// TIA Portal V20 export
DATA_BLOCK "ControlNodes"   // DB31
AUTHOR : ERsystem_FA2_DH. Kim
// stored: Access Published, MemoryReserve 100, Namespace Unit1
   VAR
      fuses { ExternalWritable := 'False'} : Struct
         motorpower_mcFeedBack : Bool;
         E202CB_motorpower_tripped : Bool;
         E208CB_maincontrol_panelMain_power_tripped : Bool;
         E320CB_E9304PWS_controlpower_SMPS_AC_power_tripped : Bool;
         E326CB_E9404PWS_controlpower_SMPS_AC_power_tripped : Bool;
         E400CB_compensator_X_Axis_power_TR_primarytripped : Bool;
         E410CB_compensator_X_Axis_power_TR_ECONDARYtripped : Bool;
         E500CB_sepa_pnp_X_Axis_powerTr_primary_tripped : Bool;
         E510CB_sepa_pnp_X_Axis_powerTr_ECONDARY_tripped : Bool;
         E720CB_powerMetrt_powerTRIIPED : Bool;
         E726CB_powerMetrt_controlpower_TRIIPED : Bool;
         E3304CB_compensator_X_Axis_power_onTrippred : Bool;
         E3504CB_sepa_pnp1_X_Axis_power_onTrippred : Bool;
         E3604CB_sepa_pnp2_X_Axis_power_onTrippred : Bool;
         E7116CB_procrssor_power_ontrippred : Bool;
         E7156CB_maincontrol_panelHot_power_tripped : Bool;
         E7304CB_panelLed_power_tripped : Bool;
         E8100CB_120VAC_control_powerTr_primary_tripped : Bool;
         E8110CB_120VAC_control_powerTr_secondary_tripped : Bool;
         E8116CB_control_power_ONtripped : Bool;
         E8156CB_maincontrol_panelControl_power_tripped : Bool;
         E9122CB_encoder_terminalUnit_control_power_tripped : Bool;
         E9128CB_servo_control_UNITcontrol_power_tripped : Bool;
         E9204CB_panelFan_power_tripped : Bool;
         E9306CB_controlDc_power_tripped : Bool;
         E9316CB_servo_control_power_tripped : Bool;
         E9406CB_controlDc_power_tripped : Bool;
         E9416CB_junctionBox_class_2SMPS_tripped : Bool;
         E9422CB_EQUIPMENT_LED_power_tripped : Bool;
         E214CB_E6404PWS_controlLER_power_SMPS_AC_power_tripped : Bool;
         E222CB_E6704PWS_controlLER_power_SMPS_AC_power_tripped : Bool;
         E226CB_E6804PWS_safety_power_SMPS_AC_power_tripped : Bool;
         E4120CB_procrssor_power_onTrpped : Bool;
         E4126CB_programing_power_outletTrpped : Bool;
         E4304CB_panelLed_power_tripped : Bool;
         E4420CB_controlLevel_hub_power_tripped : Bool;
         E4426CB_mainHmi_power_tripped : Bool;
         E4432CB_portableHmi_power_TIPPED : Bool;
         E4604CB_panelIrtHub_power_TIPPED : Bool;
         E4608ES_irtHub_fault : Bool;
         E5110CB_120VAC_control_power_TR_secondary_tripped : Bool;
         E5120CB_control_power_onTrippred : Bool;
         E5126CB_visionMonitor1_MCU_power_strip_outlet_power_tripped : Bool;
         E5132CB_visionMonitor2_visionMonitor3_power_strip_outlet_power_tripped : Bool;
         E5156CB_vision_LIGHT_controller_power_strip_outlet_power_tripped : Bool;
         E5222CB_FFU_power1_power_tripped : Bool;
         E6154CB_ET200MP_io_output_power_tripped : Bool;
         E6180CB_junctionBox_control_power_tripped : Bool;
         E6204CB_class2_SMPS_power_tripped : Bool;
         E6220CB_ET200ECO_PN1_power_tripped : Bool;
         E6224CB_ET200ECO_PN2_power_tripped : Bool;
         E6228CB_ET200ECO_PN3_power_tripped : Bool;
         E6232CB_ET200ECO_PN4_power_tripped : Bool;
         E6304CB_panelFan_power_tripped : Bool;
         E6406CB_controlLer_DC_power_tripped : Bool;
         E6422CB_mainFold1_control_power_tripped : Bool;
         E6430CB_mainFold2_control_power_tripped : Bool;
         E6456CB_driveCliq_hub_power_tripped : Bool;
         E6462CB_driveCliq_hub_power_tripped : Bool;
         E6468CB_handy_qr_reader_power_tripped : Bool;
         E6474CB_vision_controller1_power_tripped : Bool;
         E6480CB_vision_controller2_power_tripped : Bool;
         E6486CB_vision_controller3_power_tripped : Bool;
         E6506CB_linedLaser_module1_power_tripped : Bool;
         E6512CB_linedLaser_module2_power_tripped : Bool;
         E6706CB_controlLER_DC_power_tripped : Bool;
         E6716CB_EPC_controller1_power_tripped : Bool;
         E6722CB_EPC_controller2_power_tripped : Bool;
         E6728CB_EPC_controller3_power_tripped : Bool;
         E6734CB_EPC_controller4_power_tripped : Bool;
         E6806CB_safetyDc_power_tripped : Bool;
         E6816CB_ET200SP_io_safety_power_tripped : Bool;
         E6836CB_junctionBox_control_power_tripped : Bool;
         E6856CB_ET200ECO_PN_safety_1_power_tripped : Bool;
         E6862CB_ET200ECO_PN_safety_2_power_tripped : Bool;
         E6756CB_dcdc_converter_in_power_tripped : Bool;
         E6762CB_hotWire_cutter_power_tripped : Bool;
         E110CB_mainHmi_power_tripped : Bool;
      END_STRUCT;
      pws : Struct
         E9104PWS_control_power_smpSdc_ok { ExternalWritable := 'False'} : Bool;
         E9304PWS_control_power_smpSdc_ok { ExternalWritable := 'False'} : Bool;
         E9404PWS_control_power_smpSdc_ok { ExternalWritable := 'False'} : Bool;
         E4404PWS_plc_powerSmpsDc_ok : Bool;
         E6104PWS_control_powerSmpsDc_ok : Bool;
         E6206PWS_class2_smps_monitoring : Bool;
         E6404PWS_controller_powerSmpsDc_ok : Bool;
         E6704PWS_controller_powerSmpsDc_ok : Bool;
         E6804PWS_safety_powerSmpsDc_ok : Bool;
      END_STRUCT;
      motorPowerMC : Struct
         feedBack { ExternalWritable := 'False'} : Bool := FALSE;
         mcOn : Bool := FALSE;
         ready : Bool := TRUE;
         operation : Bool := FALSE;
         run : Bool := FALSE;
         fault { ExternalWritable := 'False'} : Bool := FALSE;
         error { ExternalWritable := 'False'} : Bool := FALSE;
      END_STRUCT;
      airOK { ExternalWritable := 'False'} : Bool := FALSE;   // Compressed air OK
      AutoStartEnable { ExternalWritable := 'False'} : Bool;
      InitializeEnable { ExternalWritable := 'False'} : Bool;
      BA010 { ExternalWritable := 'False'} : "LER_typeCommunicationControlNode";
      BA015 { ExternalWritable := 'False'} : "LER_typeCommunicationControlNode";
      BA060 { S7_SetPoint := 'True'} : "LER_typeCommunicationControlNode";
      BA030 { S7_SetPoint := 'True'} : "LER_typeCommunicationControlNode";
      cmFFU { S7_SetPoint := 'True'} : "LER_typeLIU117ControlNode";
      cmPowerMeter_PAC3220 { S7_SetPoint := 'True'} : "LER_typePAC3220ControlNode";
      cmHandyQRreadDM8700 { S7_SetPoint := 'True'} : "LER_typeDM8700ControlNode";
   END_VAR
BEGIN
   BA010.commands.Communication_Reset := FALSE;
   BA010.monitoring.error := FALSE;
   BA010.monitoring.status := 16#0000;
   BA015.commands.Communication_Reset := FALSE;
   BA015.monitoring.error := FALSE;
   BA015.monitoring.status := 16#0000;
   cmFFU.commands.Reset := FALSE;
   cmFFU.commands.Save := FALSE;
   cmFFU.Monitoring.RPM_PV := 1250;
   cmFFU.Monitoring.Alarm[0] := FALSE;
   cmFFU.Monitoring.Alarm[1] := TRUE;
   cmFFU.Monitoring.Alarm[2..6] := FALSE;
   cmFFU.Monitoring.Error := FALSE;
END_DATA_BLOCK
